(* IEC 61131-3 sources: CodesysTest/export/SX_1195.dev/Plc Logic/Application/PRJ Specific/1195 Testing/BagDelivery/IBagDelivery.itf, 3 files *)

(* ---- FeedAtPrintSpeed.m.st ---- *)
(*#-#-#-#-#-#-#-#-#-#---Declaration---#-#-#-#-#-#-#-#-#-#-#-#-#*)

METHOD FeedAtPrintSpeed
VAR_INPUT
END_VAR

(* ---- FeedBagOut.m.st ---- *)
(*#-#-#-#-#-#-#-#-#-#---Declaration---#-#-#-#-#-#-#-#-#-#-#-#-#*)

METHOD FeedBagOut
VAR_INPUT
END_VAR

(* ---- ReverseToSeparate.m.st ---- *)
(*#-#-#-#-#-#-#-#-#-#---Declaration---#-#-#-#-#-#-#-#-#-#-#-#-#*)

METHOD ReverseToSeparate
VAR_INPUT
	//dryCycleEnable : BOOL;
END_VAR
